{attribute 'qualified_only'}
{attribute 'strict'}
{attribute 'to_string'}
TYPE E_FilterType  :
(
   LowPass := 0,     // Low-pass filter
    HighPass := 1     // High-pass filter
);
END_TYPE

(* stored: Version 1.1.0.1
   DUT E_FilterType: Id {e713c50b-21bd-4287-985a-f12a4bdbf5a2} *)
